// TIA Portal V20 export
DATA_BLOCK "ProdDataSimulation"   // DB5
{ DB_Accessible_From_OPC_UA := 'FALSE' }
// stored: DBAccessibleFromOPCUA false, DBAccessibleFromWebserver false, MemoryReserve 100
   VAR
      ProdDataCounter { ExternalAccessible := 'False'; ExternalVisible := 'False'; ExternalWritable := 'False'} : Struct   // Test tag prod data
         ProdDataCounter1Up1 : Bool := FALSE;   // Test Variable Prod. Daten / Test tag prod data
         ProdDataCounter1Up2 : Bool := FALSE;   // Test Variable Prod. Daten / Test tag prod data
         ProdDataCounter1Down1 : Bool := FALSE;   // Test Variable Prod. Daten / Test tag prod data
         ProdDataCounter1Down2 : Bool := FALSE;   // Test Variable Prod. Daten / Test tag prod data
         ProdDataCounter1Reset1 : Bool := FALSE;   // Test Variable Prod. Daten / Test tag prod data
         ProdDataCounter1Reset2 : Bool := FALSE;   // Test Variable Prod. Daten / Test tag prod data
         ProdDataCounter1ResetAll : Bool := FALSE;   // Test Variable Prod. Daten / Test tag prod data
         ProdDataCounter2Up1 : Bool := FALSE;
         ProdDataCounter2Up2 : Bool := FALSE;
         ProdDataCounter2Down1 : Bool := FALSE;
         ProdDataCounter2Down2 : Bool := FALSE;
         ProdDataCounter2Reset1 : Bool := FALSE;
         ProdDataCounter2Reset2 : Bool := FALSE;
         ProdDataCounter2ResetAll : Bool := FALSE;
         userInterfaceVisibilityDataSet2Counter : DWord := 16#000F_FFFF;
         userInterfaceVisibilityDataSet1Counter : DWord := 16#0000_3FFF;
         ProdDataEnable : Bool := FALSE;
      END_STRUCT;
      ProdDataCyclic { ExternalAccessible := 'False'; ExternalVisible := 'False'; ExternalWritable := 'False'} : Struct   // Test tag prod data
         cycleTimer1Run1 : Bool := FALSE;   // Test Variable Prod. Daten / Test tag prod data
         cycleTimer1Run2 : Bool := FALSE;   // Test Variable Prod. Daten / Test tag prod data
         cycleTimer1Hold1 : Bool := FALSE;   // Test Variable Prod. Daten / Test tag prod data
         cycleTimer1Hold2 : Bool := FALSE;   // Test Variable Prod. Daten / Test tag prod data
         cycleTimer1Reset1 : Bool := FALSE;   // Test Variable Prod. Daten / Test tag prod data
         cycleTimer1Reset2 : Bool := FALSE;   // Test Variable Prod. Daten / Test tag prod data
         cycleTimer1ResetAll : Bool := FALSE;   // Test Variable Prod. Daten / Test tag prod data
         cycleTimer2Run1 : Bool := FALSE;   // Test Variable Prod. Daten / Test tag prod data
         cycleTimer2Run2 : Bool := FALSE;   // Test Variable Prod. Daten / Test tag prod data
         cycleTimer2Hold1 : Bool := FALSE;   // Test Variable Prod. Daten / Test tag prod data
         cycleTimer2Hold2 : Bool := FALSE;   // Test Variable Prod. Daten / Test tag prod data
         cycleTimer2Reset1 : Bool := FALSE;   // Test Variable Prod. Daten / Test tag prod data
         cycleTimer2Reset2 : Bool := FALSE;   // Test Variable Prod. Daten / Test tag prod data
         cycleTimer2ResetAll : Bool := FALSE;   // Test Variable Prod. Daten / Test tag prod data
         cyclicTimerEnable : Bool := FALSE;
         userInterfaceVisibilityDataSet1Cyclic : DWord := 2#0000_0000_0000_0000_0000_0010_0000_0011;
         userInterfaceVisibilityDataSet2Cyclic : DWord := 2#0000_0000_0000_0000_0000_0010_0000_0011;
         userInterfaceVisibilityDataSet3Cyclic : DWord := 2#0000_0000_0000_0000_0000_0010_0000_0011;
         userInterfaceVisibilityDataSet4Cyclic : DWord := 2#0000_0000_0000_0000_0000_0000_0000_0011;
         userInterfaceVisibilityDataSet5Cyclic : DWord := 2#0000_0000_0000_0001_1111_1111_1011_1111;
         userInterfaceVisibilityDataSet6Cyclic : DWord := 2#0000_0000_0000_0001_1111_1111_1011_1111;
         userInterfaceVisibilityDataSet7Cyclic : DWord := 2#0000_0000_0000_0101_0011_1100_1100_1011;
         userInterfaceVisibilityDataSet8Cyclic : DWord := 2#0000_0000_0000_0000_1111_1101_1111_0111;
      END_STRUCT;
      ProdDataLimitValues { ExternalAccessible := 'False'; ExternalVisible := 'False'; ExternalWritable := 'False'} : Struct   // Test tag prod data
         limitVal1Count1PreWarn1 : Bool := FALSE;   // Test Variable Prod. Daten / Test tag prod data
         limitVal1Count1PreWarn3 : Bool := FALSE;   // Test Variable Prod. Daten / Test tag prod data
         limitVal1Count1PreWarn2 : Bool := FALSE;   // Test Variable Prod. Daten / Test tag prod data
         limitVal1Count1Alarm1 : Bool := FALSE;   // Test Variable Prod. Daten / Test tag prod data
         limitVal1Count1Alarm3 : Bool := FALSE;   // Test Variable Prod. Daten / Test tag prod data
         limitVal1Count1Alarm2 : Bool := FALSE;   // Test Variable Prod. Daten / Test tag prod data
         limitVal1Count1 : Bool := FALSE;   // Test Variable Prod. Daten / Test tag prod data
         limitVal1Count2 : Bool := FALSE;   // Test Variable Prod. Daten / Test tag prod data
         limitVal1Count3 : Bool := FALSE;   // Test Variable Prod. Daten / Test tag prod data
         limitVal1Set1 : Bool := FALSE;   // Test Variable Prod. Daten / Test tag prod data
         limitVal1Set3 : Bool := FALSE;   // Test Variable Prod. Daten / Test tag prod data
         limitVal1Set2 : Bool := FALSE;   // Test Variable Prod. Daten / Test tag prod data
         limitValuesEnable : Bool := FALSE;
         userInterfaceVisibilityDataSet2LimitValues : DWord := 16#0000_03FF;
         userInterfaceVisibilityDataSet1LimitValues : DWord := 16#0000_000F;
      END_STRUCT;
      ProdDataShiftCounter { ExternalAccessible := 'False'; ExternalVisible := 'False'; ExternalWritable := 'False'} : Struct   // Test tag prod data
         shiftCounter1Cnt1Curr : Bool := FALSE;   // Test Variable Prod. Daten / Test tag prod data
         shiftCounter1Cnt1CurrOk : Bool := FALSE;   // Test Variable Prod. Daten / Test tag prod data
         shiftCounter1Cnt2Curr : Bool := FALSE;   // Test Variable Prod. Daten / Test tag prod data
         shiftCounter1Cnt2CurrOk : Bool := FALSE;   // Test Variable Prod. Daten / Test tag prod data
         shiftCounter1Cnt3Curr : Bool := FALSE;   // Test Variable Prod. Daten / Test tag prod data
         shiftCounter1Cnt3CurrOk : Bool := FALSE;   // Test Variable Prod. Daten / Test tag prod data
         shiftCounter1ResetAllExt : Bool := FALSE;   // Test Variable Prod. Daten / Test tag prod data
         ShiftCounterEnable : Bool := FALSE;
         userInterfaceVisibilityDataSet2ShiftCounter : DWord := 16#0000_03FF;
         userInterfaceVisibilityDataSet1ShiftCounter : DWord := 16#0000_000F;
      END_STRUCT;
      ProdDataShiftCounterOEE { ExternalAccessible := 'False'; ExternalVisible := 'False'; ExternalWritable := 'False'} : Struct   // Test tag prod data
         ShiftCounterOEEEnable : Bool := FALSE;
         userInterfaceVisibilityDataSet2ShiftCounterOEE : DWord := 16#0000_03FF;
         userInterfaceVisibilityDataSet1ShiftCounterOEE : DWord := 16#0000_000F;
      END_STRUCT;
   END_VAR
BEGIN
END_DATA_BLOCK
